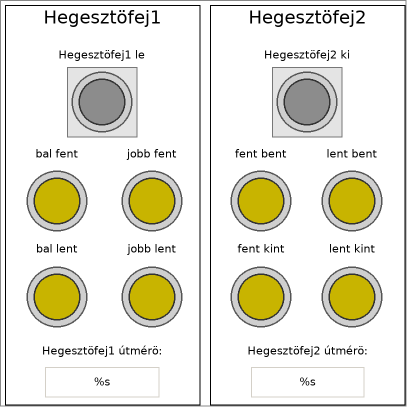
VISUALIZATION Hegesztofej_IOk_NTC  // 407x407
    Group (5,5 195x400)
        Rectangle (0,0 195x400), "Hegesztöfej1"
        Textfield (40,362 114x30), "%s", text variable: HEGESZTOK.ulHegeszto1Utmero, input disabled if: TRUE
        Label (34,336 126x20), "Hegesztöfej1 útmérö:"
        Lamp1 (17,161 70x70), variable: GVL.bHegeszto1BalFent, style: Lamp-Lamp1-Yellow
        Label (22,139 60x20), "bal fent"
        Lamp1 (17,257 70x70), variable: GVL.bHegeszto1BalLent, style: Lamp-Lamp1-Yellow
        Label (22,234 60x20), "bal lent"
        Lamp1 (112,161 70x70), variable: GVL.bHegeszto1JobbFent, style: Lamp-Lamp1-Yellow
        Label (117,139 60x20), "jobb fent"
        Lamp1 (112,257 70x70), variable: GVL.bHegeszto1JobbLent, style: Lamp-Lamp1-Yellow
        Label (117,234 60x20), "jobb lent"
        PushSwitch (62,62 70x70), variable: HEGESZTOK.bHegesztoFejekOutput[0], behaviour: TOGGLE, style: Switch-PushSwitch-Gray
        Label (39,40 116x20), "Hegesztöfej1 le"
    Group (210,5 195x400)
        Rectangle (0,0 195x400), "Hegesztöfej2"
        Textfield (41,362 113x30), "%s", text variable: HEGESZTOK.ulHegeszto2Utmero, input disabled if: TRUE
        Label (33,336 129x20), "Hegesztöfej2 útmérö:"
        Lamp1 (16,257 70x70), variable: GVL.bHegeszto2FentKint, style: Lamp-Lamp1-Yellow
        Label (21,234 60x20), "fent kint"
        Lamp1 (16,161 70x70), variable: GVL.bHegeszto2FentBent, style: Lamp-Lamp1-Yellow
        Label (21,139 60x20), "fent bent"
        Lamp1 (107,257 70x70), variable: GVL.bHegeszto2LentKint, style: Lamp-Lamp1-Yellow
        Label (112,234 60x20), "lent kint"
        Lamp1 (107,161 70x70), variable: GVL.bHegeszto2LentBent, style: Lamp-Lamp1-Yellow
        Label (112,139 60x20), "lent bent"
        Label (39,40 116x20), "Hegesztöfej2 ki"
        PushSwitch (62,62 70x70), variable: HEGESZTOK.bHegesztoFejekOutput[1], behaviour: TOGGLE, style: Switch-PushSwitch-Gray
END_VISUALIZATION

(* stored: Version 1.1.0.1, ProductVersion 3.1.4024.11
   Visu Hegesztofej_IOk_NTC: Id {b6551e4b-0021-4865-98b9-c0a68d8fb39f} *)
